FUNCTION_BLOCK FLOW_METER
VAR_INPUT
	VX : REAL;
	E : BOOL;
	RST : BOOL;
END_VAR
VAR_INPUT CONSTANT
	PULSE_MODE : BOOL;
	UPDATE_TIME : TIME := t#1s;
END_VAR
VAR_OUTPUT
	F : REAL;
END_VAR
VAR_IN_OUT
	X : REAL;
	Y : UDINT;
END_VAR
VAR
	tx, tl : TIME;
	int1 : INTEGRATE;
	init: BOOL;
	e_last : BOOL;
	tmp: INT;
	x_last : REAL;
	y_last : UDINT;
END_VAR

(*
version 1.0	23. jan. 2011
programmer 	hugo
tested by	oscat

Flow meter measures flow according to gated time or pulses.

*)

IF NOT init THEN	(* init on power up *)
	init := TRUE;
	tl := tx;
	x_last := X;
	y_last := Y;
	int1.K := 2.7777777777777777E-4;
END_IF;

(* run integrator *)
int1(E := NOT (RST OR PULSE_MODE) AND E, X := VX, Y := X);	(* gated operation *)

IF RST THEN		(* reset *)
	X := 0.0;
	Y := 0;
	tl := tx;
	x_last := 0.0;
	y_last := 0;
ELSIF E AND PULSE_MODE THEN	(* check for pulse mode *)
	IF NOT e_last THEN X := X + VX; END_IF;
END_IF;
e_last := E;

(* reduce X to be less than 1 and increase Y respectively *)
IF X > 1.0 THEN
	tmp := FLOOR(X);
	Y := Y + INT_TO_UDINT(tmp);
	X := X - INT_TO_REAL(tmp);
END_IF;

(* calculate the current flow *)
tx := DWORD_TO_TIME(T_PLC_MS());
IF tx - tl >= UPDATE_TIME AND UPDATE_TIME > t#0s THEN
	F := (UDINT_TO_REAL(Y - y_last) + X - x_last) / TIME_TO_REAL(tx - tl) * 3.6E6;
	y_last := Y;
	x_last := X;
	tl := tx;
END_IF;



(* revision history
hm	23. jan. 2011	rev 1.0
	original version

*)

END_FUNCTION_BLOCK

(* stored: Version 1.1.0.1, ProductVersion 3.1.4022.7
   POU FLOW_METER: Id {c4fed62f-7891-419a-9837-7ecf59458acb}, SpecialFunc None *)
